_CFC_ (* Continuous Function Chart, elements in execution order *)
#0 SEL(#14, #6, eHVAC2PointActuatorMode_Close_OP)
#1 ZADERJ_SHOD_YA1:TON(IN: #5.Q1, PT: t#10s)
#2 RT_Pusk:R_TRIG(CLK: SCHU_P2_2_UST_RE_PUSK)
#3 TON_PCH_OTKL:TON(IN: SCHU_P2_2_UST_RE_STOP, PT: T#1s)
#4 FT_PCH_OTKL:R_TRIG(CLK: #3.Q)
#5 RS_YA1_Open:RS(SET: #2.Q, RESET1: #4.Q)
#6 SEL(SCHU_P2_2_SA7_DI1_A, eHVAC2PointActuatorMode_Close_OP, eHVAC2PointActuatorMode_Auto_BMS)
#7 fb_HVACPA:FB_HVAC2PointActuator(eHVACDataSecurityType_Idle, FALSE, TRUE, #1.Q, #0, SCHU_P2_2_KV1_DI4, SCHU_P2_2_YA1_DI6_ZKR, SCHU_P2_2_YA1_DI7_OTK, TRUE, SCHU_P2_2_SB, enableLimitSwitch, stokeTime)
#8 SCHU_P2_2_SA7_DO7_OTK <= #7.out 1
#9 OR(#7.out 4, #7.out 5)
#10 YA1_OTKAZ <= #9
#11 INT_TO_TIME(SCHU_P2_2_YA1_VREMYA_HODA)
#12 MUL(#11, 1000)
#13 stokeTime <= #12
#14 OR(#15.Q, Z_ZAM_SR)
#15 TON_YA1_Z_ZAM_TE2:TON(IN: SCHU_P2_2_TE2_M_ZASCH, PT: t#5s)
_END_CFC_
END_PROGRAM

(* POU IM/YA2_Upr, CFC *)
PROGRAM YA2_Upr
VAR
	YA2_PID: FB_HVACPIDCtrl;

	deadRange: REAL := 0.1;
	direction: BOOL;
	tTi: TIME;
	tTv: TIME;
	tTd: TIME;

	rYMin: REAL := 0;
	rYMax: REAL := 100;
	TON_SCHU_P2_2_P1_DI4_RUN: TON;
	reg1: BOOL;
	reg2: BOOL;

	SCHU_P2_2_YA2_: BOOL;
	YA2_REG_POL: BOOL;
	rwx: REAL;
	EPS1: REAL;
	EPS2: REAL;
END_VAR
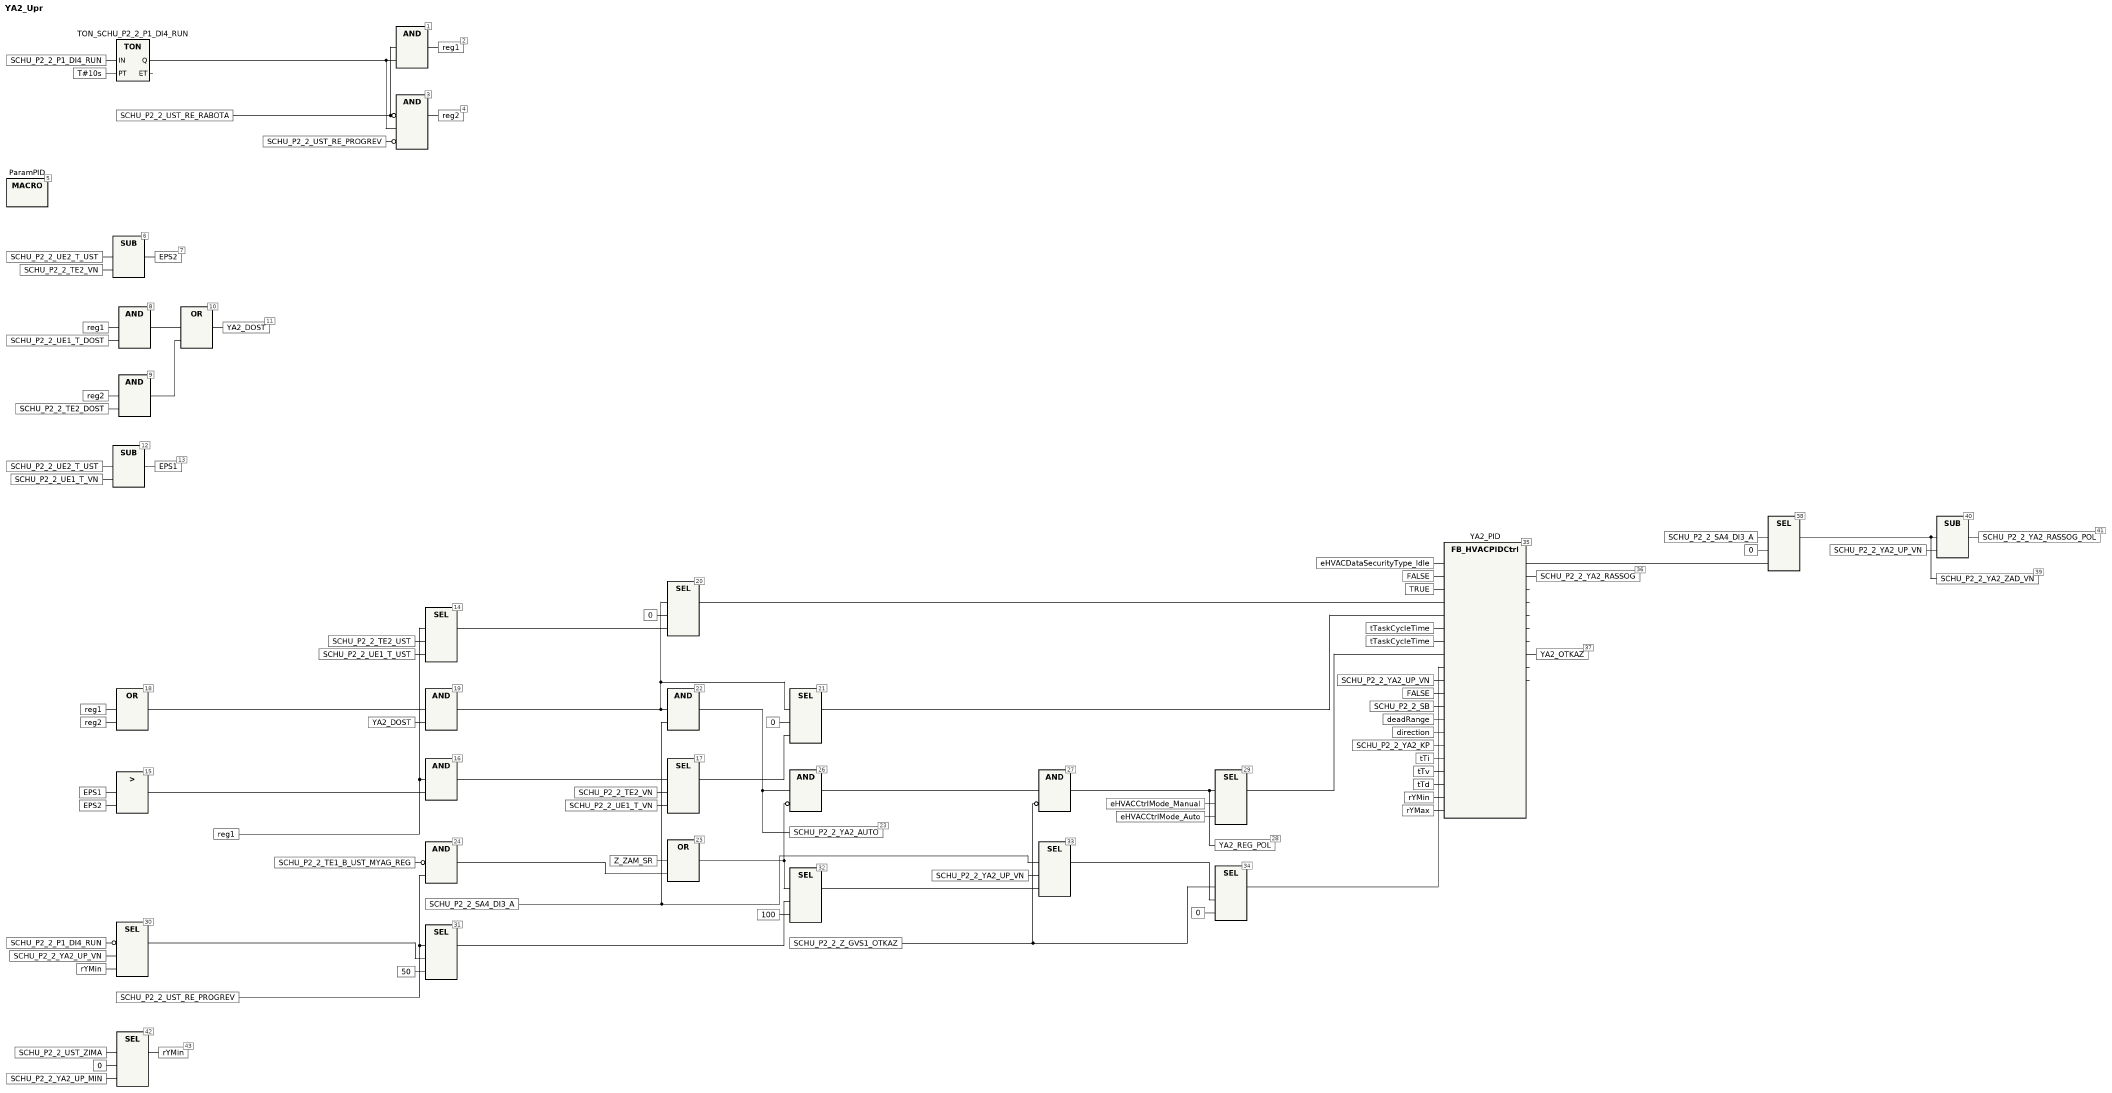
